TYPE Cnv_VTD_Settings_DUT :
STRUCT
	Cnv_Level:	ARRAY[2..6] OF Cnv_Level_Settings_DUT;
END_STRUCT
END_TYPE

(* stored: Version 1.1.0.1
   DUT Cnv_VTD_Settings_DUT: Id {fc1c9d53-18ce-4be4-a3a1-609f9673e009} *)
